TYPE ST_LaudaReadCommands_Rights :
STRUCT
	KeyboardMaster_Locked				: STRING := 'IN_MODE_00_';
	KeyboardRemoveControlUnit_Locked	: STRING := 'IN_MODE_03';
END_STRUCT
END_TYPE

(* stored: Version 1.1.0.1, ProductVersion 3.1.4024.12
   DUT ST_LaudaReadCommands_Rights: Id {ea0401cc-c3df-443a-8a40-289bca2fadcc} *)
